PROGRAM MAIN
VAR
END_VAR

END_PROGRAM

(* stored: Version 1.1.0.1
   POU MAIN: Id {db1d7828-d60e-431f-b43a-c5c356d1b311} *)
